// TIA Portal V18 export
FUNCTION "DIbasic" : Void   // FC10003, LAD
{ S7_Optimized_Access := 'TRUE' }
VERSION : 0.1
// stored: AutoNumber false, IsIECCheckEnabled false, SetENOAutomatically false, UDAEnableTagReadback false
   VAR_INPUT
      xInput : Bool;
      xInversion : Bool;   // 0-direct / 1-reverse
   END_VAR
   VAR_OUTPUT
      xOutputFiltered : Bool;
   END_VAR
   VAR_IN_OUT
      iAddImpOff : Int;
      xMemory : Bool;
      iAddImpOn : Int;
      iCounter : Int;
   END_VAR
   VAR_TEMP
      InOut_1 : Bool;
   END_VAR
   VAR_TEMP   // added for the SCL form of the ladder/FBD networks
      _w1 : Bool;
      _w2 : Bool;
   END_VAR
BEGIN

REGION Network 1 (FBD)
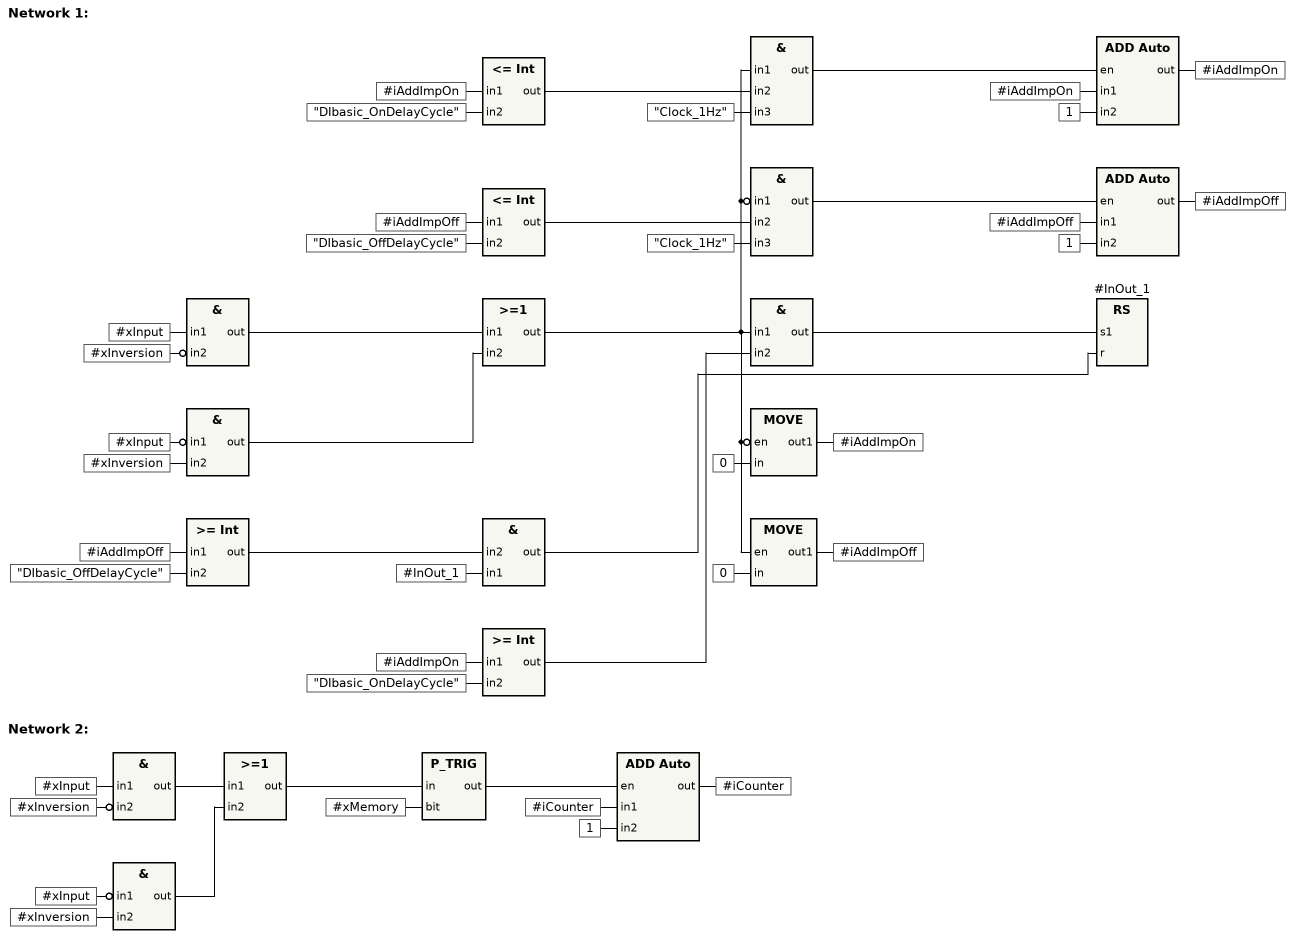
   #_w1 := (#xInput AND NOT #xInversion) OR (NOT #xInput AND #xInversion);
   IF #_w1 AND (#iAddImpOn <= "DIbasic_OnDelayCycle") AND "Clock_1Hz" THEN
       #iAddImpOn := #iAddImpOn + 1;
   END_IF;
   IF NOT #_w1 AND (#iAddImpOff <= "DIbasic_OffDelayCycle") AND "Clock_1Hz" THEN
       #iAddImpOff := #iAddImpOff + 1;
   END_IF;
   IF (#iAddImpOff >= "DIbasic_OffDelayCycle") AND #InOut_1 THEN
       #InOut_1 := FALSE;   // RS flip-flop
   END_IF;
   IF #_w1 AND (#iAddImpOn >= "DIbasic_OnDelayCycle") THEN #InOut_1 := TRUE; END_IF;
   IF NOT #_w1 THEN #iAddImpOn := 0; END_IF;
   IF #_w1 THEN #iAddImpOff := 0; END_IF;
END_REGION

REGION Network 2 (FBD)
   #_w1 := (#xInput AND NOT #xInversion) OR (NOT #xInput AND #xInversion);
   #_w2 := #_w1 AND NOT #xMemory;   // rising edge
   #xMemory := #_w1;
   IF #_w2 THEN #iCounter := #iCounter + 1; END_IF;
END_REGION

REGION Network 3
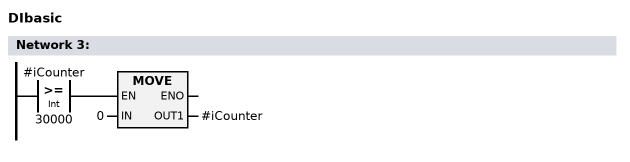
   RUNG wire#powerrail
      { S7_Templates := "SrcType := Int" } GE_Contact(in1 := #iCounter, in2 := 30000)
      Move(in := 0, out1 => #iCounter)
   END_RUNG
   // the same network as SCL:
   IF #iCounter >= 30000 THEN #iCounter := 0; END_IF;
END_REGION
END_FUNCTION
